{attribute 'GeneratedUsingTerminal: AX8108-0100-0101-0101'}
{attribute addProperty BoxType "AX8108-0100-0101-0101"}
{attribute addProperty Id "FSoE_Slave_CmdUSINT1Axis_A_STOBOOL1Safe_Input_1BOOL1Safe_Input_2BOOL1Safe_Input_3BOOL1Safe_Input_4BOOL1Safe_Input_5BOOL1Safe_Input_6BOOL1Safe_Input_7BOOL1Axis_B_STOBOOL1Safe_Input_9BOOL1Safe_Input_10BOOL1Safe_Input_11BOOL1Safe_Input_12BOOL1Safe_Input_13BOOL1Safe_Input_14BOOL1Safe_Input_15BOOL1FSoE_Slave_CRC_0UINT2FSoE_Slave_ConnIDUINT2"}
{attribute addProperty CRC "834371370"}
{attribute addProperty Size "21"}
TYPE FSOE_31BB7F2A :
STRUCT
	{attribute addProperty Name "FSoE_Slave_Cmd"}
	FSoE_Slave_Cmd : USINT;
	{attribute addProperty Name "Axis_A_STO"}
	Axis_A_STO : BOOL;
	{attribute addProperty Name "Safe_Input_1"}
	Safe_Input_1 : BOOL;
	{attribute addProperty Name "Safe_Input_2"}
	Safe_Input_2 : BOOL;
	{attribute addProperty Name "Safe_Input_3"}
	Safe_Input_3 : BOOL;
	{attribute addProperty Name "Safe_Input_4"}
	Safe_Input_4 : BOOL;
	{attribute addProperty Name "Safe_Input_5"}
	Safe_Input_5 : BOOL;
	{attribute addProperty Name "Safe_Input_6"}
	Safe_Input_6 : BOOL;
	{attribute addProperty Name "Safe_Input_7"}
	Safe_Input_7 : BOOL;
	{attribute addProperty Name "Axis_B_STO"}
	Axis_B_STO : BOOL;
	{attribute addProperty Name "Safe_Input_9"}
	Safe_Input_9 : BOOL;
	{attribute addProperty Name "Safe_Input_10"}
	Safe_Input_10 : BOOL;
	{attribute addProperty Name "Safe_Input_11"}
	Safe_Input_11 : BOOL;
	{attribute addProperty Name "Safe_Input_12"}
	Safe_Input_12 : BOOL;
	{attribute addProperty Name "Safe_Input_13"}
	Safe_Input_13 : BOOL;
	{attribute addProperty Name "Safe_Input_14"}
	Safe_Input_14 : BOOL;
	{attribute addProperty Name "Safe_Input_15"}
	Safe_Input_15 : BOOL;
	{attribute addProperty Name "FSoE_Slave_CRC_0"}
	FSoE_Slave_CRC_0 : UINT;
	{attribute addProperty Name "FSoE_Slave_ConnID"}
	FSoE_Slave_ConnID : UINT;
END_STRUCT
END_TYPE

(* stored: Version 1.2.0.0, ProductVersion 3.1.4024.9
   DUT FSOE_31BB7F2A: Id {5361c0ca-81d2-4612-a271-194f7b292f4b} *)
